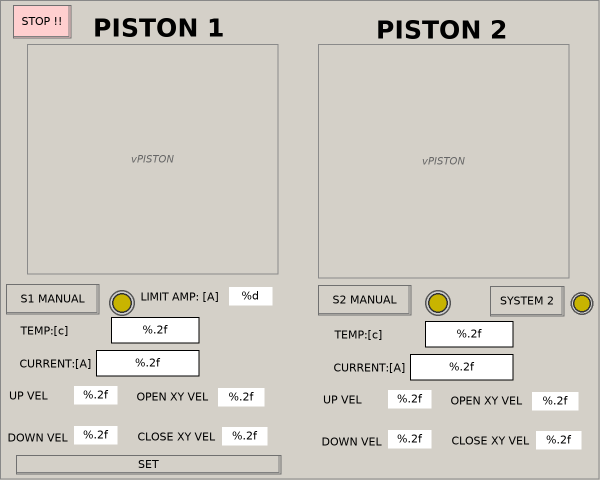
VISUALIZATION vPISTONS  // 600x480
    Frame (318,44 251x234), invisible if: true
        shows vPISTON(PIST1 := PIST2, MANUAL := ACTION2.bMANUAL)
    Frame (27,44 251x230)
        shows vPISTON(PIST1 := PIST1, MANUAL := ACTION1.bMANUAL)
    Label (84,14 150x27), "PISTON 1"
    Label (367,16 150x27), "PISTON 2", invisible if: true
    Button (490,286 74x30), "SYSTEM 2", invisible if: true
        toggle bSECOND_SYS
    Label (-17,385 91x22), "UP VEL"
    Label (-8,427 91x22), "DOWN VEL"
    Textfield (73,425 45x20), "%.2f", text variable: LIFT1_DOWN_VEL
        OnMouseDown: write the text variable via Default
    Textfield (217,387 48x20), "%.2f", text variable: XY1_OPEN_VEL
        OnMouseDown: write the text variable via Default
    Label (127,386 91x22), "OPEN XY VEL"
    Textfield (221,426 47x20), "%.2f", text variable: XY1_CLOSE_VEL
        OnMouseDown: write the text variable via Default
    Label (131,426 91x22), "CLOSE XY VEL"
    Label (77,297 91x22)
    Label (358,297 91x22)
    Rectangle (111,317 88x26), "%.2f", text variable: ACTION1.iTEMP_SHOW
    Rectangle (96,350 103x26), "%.2f", text variable: ACTION1.iCURRENT_PISTON_SHOW
    Label (18,320 53x22), "TEMP:[c]"
    Label (10,353 91x22), "CURRENT:[A]"
    Button (6,284 93x30), "S1 MANUAL"
        OnMouseDown: execute { ACTION1.bMANUAL:=TRUE; }
    Lamp1 (107,285 30x36), variable: ACTION1.bMANUAL, style: Lamp-Lamp1-Yellow
    Button (318,285 93x30), "S2 MANUAL", invisible if: true, input disabled if: NOT ACTION2.bALL_HOMED
        OnMouseDown: execute { ACTION2.bMANUAL:=TRUE; }
    Lamp1 (423,285 30x36), variable: ACTION2.bMANUAL, invisible if: true, style: Lamp-Lamp1-Yellow
    Lamp1 (569,288 26x31), variable: bSECOND_SYS, invisible if: true, style: Lamp-Lamp1-Yellow
    Button (13,5 58x33), "STOP !!"
        OnMouseDown: execute { ACTION1.bSTOP_ALL:=TRUE; }
    Textfield (73,385 45x20), "%.2f", text variable: LIFT1_UP_VEL
        OnMouseDown: write the text variable via Default
    Button (16,455 265x19), "SET"
        tap bWP_Start
    Label (138,286 84x22), "LIMIT AMP: [A]"
    Textfield (228,286 45x20), "%d", text variable: SAFETY_LIMIT1
        OnMouseDown: write the text variable via Default
    Label (297,389 91x22), "UP VEL", invisible if: true
    Label (306,431 91x22), "DOWN VEL", invisible if: true
    Textfield (387,429 45x20), "%.2f", text variable: LIFT2_DOWN_VEL, invisible if: true
        OnMouseDown: write the text variable via Default
    Textfield (531,391 48x20), "%.2f", text variable: XY2_OPEN_VEL, invisible if: true
        OnMouseDown: write the text variable via Default
    Label (441,390 91x22), "OPEN XY VEL", invisible if: true
    Textfield (535,430 47x20), "%.2f", text variable: XY2_CLOSE_VEL, invisible if: true
        OnMouseDown: write the text variable via Default
    Label (445,430 91x22), "CLOSE XY VEL", invisible if: true
    Rectangle (425,321 88x26), "%.2f", text variable: ACTION1.iTEMP_SHOW, invisible if: true
    Rectangle (410,354 103x26), "%.2f", text variable: ACTION1.iCURRENT_PISTON_SHOW, invisible if: true
    Label (332,324 53x22), "TEMP:[c]", invisible if: true
    Label (324,357 91x22), "CURRENT:[A]", invisible if: true
    Textfield (387,389 45x20), "%.2f", text variable: LIFT2_UP_VEL, invisible if: true
        OnMouseDown: write the text variable via Default
END_VISUALIZATION

(* stored: Version 1.1.0.1, ProductVersion 3.1.4024.12
   Visu vPISTONS: Id {f994902e-2012-4350-af9d-36cdf7c7a690} *)
